{attribute 'qualified_only'}
VAR_GLOBAL CONSTANT
	buffersize_filter :UINT :=2000;
END_VAR

(* stored: Version 1.1.0.1, ProductVersion 3.1.4024.13
   GVL GVL_SensorFusion: Id {04dd9f49-f948-4283-b0bc-ee4d4fa77983} *)
